// TwinCAT 3 PLC project Punzonatrice_2223
// ProgramVersion: 3.1.4024.0
// libraries:
//   Tc2_Standard, * (Beckhoff Automation GmbH)
//   Tc2_System, * (Beckhoff Automation GmbH)
//   Tc3_Module, * (Beckhoff Automation GmbH)
// project tree:
//   GVLs/ GVL_HMI.TcGVL (not stored), GVL_IO.TcGVL (not stored)
//   / PlcTask.TcTTO (not stored)
//   POUs/ FB_MSF.TcPOU, FB_Oscillatore.TcPOU, MAIN.TcPOU

// ---- POUs/FB_MSF.TcPOU
FUNCTION_BLOCK FB_MSF
VAR_INPUT
	start	:	BOOL;
	stop	:	BOOL;
	ack		:	BOOL;
	emerg	:	BOOL;
	i1		:	BOOL;
	i2		:	BOOL;
	i3		:	BOOL;
	i4		:	BOOL;
END_VAR
VAR_OUTPUT
	q1		:	BOOL;
	q2		:	BOOL;
	q3		:	BOOL;
	q4		:	BOOL;
	lstart	:	BOOL;
	lstop	:	BOOL;
	lack	:	BOOL;
END_VAR
VAR
	// enumeratore privato degli stati, la variabile stato parte da S0
	stato : (S0, S1, S2, S3, S4, S5, S6, S7, S8, SE, SA) := S0;
	
	// timer T34 attesa dopo caricamento
	T34		:	TON();
	T82		:	TON();
	
	// lampeggiatore
	osc	:	FB_Oscillatore();
	
	// bit di abilitazione
	enable	:	BOOL;
	
	// bit delle transizioni
	tr_01	:	BOOL;
	tr_02	:	BOOL;
	tr_12	:	BOOL;
	tr_23	:	BOOL;
	tr_34	:	BOOL;
	tr_45	:	BOOL;
	tr_56	:	BOOL;
	tr_67	:	BOOL;
	tr_78	:	BOOL;
	tr_80	:	BOOL;
	tr_82	:	BOOL;
	tr_EA	:	BOOL;
	tr_A0	:	BOOL;
	
	// memoria dello stop nominale
	mArresto:	BOOL := FALSE;
	
	// memoria di un pezzo in lavorazione sul nastro
	mPezzoCarico	:	BOOL := FALSE;
	
END_VAR

// 1. aggiornamento condizioni di abilitazione
enable := stop AND emerg;

// 2. aggiornamento di timers, contatori, triggers sui fronti
T34(IN := (stato = S3 AND enable), PT := T#2S );
T82(IN := (stato = S8 AND enable), PT := T#3S );
osc(enable := (stato = SA) OR (stato = SE), t_high := T#500MS, t_low := T#500MS);

// 3. condizione di arresto nominale
IF NOT stop AND emerg THEN
	IF (stato = S1 OR stato = S2) THEN
		stato := S0;
	ELSIF (stato = S3 OR stato = S4 OR stato = S5 OR stato = S6 OR stato = S7 OR stato = S8) THEN
		mArresto := TRUE;
	END_IF
END_IF

// 4. condizione di arresto di emergenza
IF NOT emerg THEN
	stato := SE;
END_IF

// 5. aggiornamento delle condizioni di transizione
tr_01 := NOT(i3) AND start AND enable;
tr_02 := i3 AND start AND enable;
tr_12 := i3 AND enable; 
tr_23 := enable AND NOT(i1);
tr_34 := enable AND NOT(i1) AND T34.Q;
tr_45 := NOT(i2) AND enable;
tr_56 := enable AND i4;
tr_67 := enable AND i3;
tr_78 := enable AND NOT(i1);
tr_80 := enable AND mArresto;
tr_82 := enable AND NOT(mArresto) AND i1 AND T82.Q;
tr_EA := emerg AND ack;
tr_A0 := (mPezzoCarico AND NOT(i1) AND i3) OR (NOT(mPezzoCarico) AND i3);

// 6. switch-case della MSF
CASE stato OF
S0:
	mArresto := FALSE;
	mPezzoCarico := FALSE;
    IF tr_02 THEN
    	stato := S2;
    ELSIF tr_01 THEN
		stato := S1;
    END_IF	
	
S1:
	IF tr_12 THEN
		stato := S2;
	END_IF

S2:
	mPezzoCarico := FALSE;
	IF tr_23 THEN
		stato := S3;
	END_IF

S3:
	mPezzoCarico := TRUE;
	IF tr_34 THEN
		stato := S4;
	END_IF	

S4:
	IF tr_45 THEN
		stato := S5;
	END_IF
	
S5:
	IF tr_56 THEN
		stato := S6;
	END_IF

S6:
	IF tr_67 THEN
		stato := S7;
	END_IF

S7:
	IF tr_78 THEN
		stato := S8;
	END_IF

S8:
	IF tr_80 THEN
    	stato := S0;
    ELSIF tr_82 THEN
		stato := S2;
    END_IF

SE:
	IF tr_EA THEN
		stato := SA;
	END_IF

SA:
	IF tr_A0 THEN
		stato := S0;
	END_IF

ELSE
	// fail over: la variabile di stato è danneggiata, vai in SE
	stato := SE;	
	
END_CASE

// 7. comando uscite
lstart := (stato <> S0);
lstop := (stato = S0) OR ((stato = SE) AND osc.Q);
lack := (stato = SE) OR ((stato = SA) AND osc.Q);
q1 := (stato = S4);
q2 := (stato = S7) OR ((stato = SA) AND mPezzoCarico);
q3 := (stato = S1) OR (stato = S6) OR ((stato = SA) AND NOT(i3));
q4 := (stato = S5);

END_FUNCTION_BLOCK

// ---- POUs/FB_Oscillatore.TcPOU
FUNCTION_BLOCK FB_Oscillatore
VAR_INPUT
	enable : BOOL;
	t_high : TIME;
	t_low : TIME;
END_VAR
VAR_OUTPUT
	q : BOOL;
END_VAR
VAR
	t1 : TON();
	t2 : TON();
END_VAR

t1(in := enable AND NOT t2.Q, pt := t_low);
t2(in := t1.Q, pt := t_high);
q := t1.Q;

END_FUNCTION_BLOCK

// ---- POUs/MAIN.TcPOU
PROGRAM MAIN
VAR
	punzonatrice	:	FB_MSF();
END_VAR

// eseguo l'istanza della punzonatrice
punzonatrice(
	start:= GVL_IO.PSTART, 
	stop:= GVL_IO.PSTOP, 
	ack:= GVL_IO.PACK, 
	emerg:= GVL_IO.PEMERG, 
	i1:= GVL_IO.I1, 
	i2:= GVL_IO.I2, 
	i3:= GVL_IO.I3, 
	i4:= GVL_IO.I4, 
	q1=> GVL_IO.Q1, 
	q2=> GVL_IO.Q2, 
	q3=> GVL_IO.Q3, 
	q4=> GVL_IO.Q4, 
	lstart=> GVL_IO.LSTART, 
	lstop=> GVL_IO.LSTOP, 
	lack=> GVL_IO.LACK);

END_PROGRAM
